// TwinCAT 3 PLC project Tc3_Handler
// ProgramVersion: 3.1.4024.0
// libraries:
//   Tc2_Standard, * (Beckhoff Automation GmbH)
//   Tc2_System, * (Beckhoff Automation GmbH)
//   Tc2_Utilities, * (Beckhoff Automation GmbH)
//   Tc3_Module, * (Beckhoff Automation GmbH)
// project tree:
//   / GVL.TcGVL (not stored), PlcTask.TcTTO
//   Library/Event/ E_Event.TcDUT, FB_Event.TcPOU, I_Event.TcIO, ST_Event.TcDUT
//   Library/Handler/ FB_Handler.TcPOU, I_Handler.TcIO
//   POUs/ FB_EventHandler.TcPOU, FB_EmergencyHandler.TcPOU, MAIN.TcPOU
// real-time tasks:
//   TASK PlcTask: cycle T#10ms, priority 20, ADS port 350

CONFIGURATION Tc3_Handler
    RESOURCE PLC ON TwinCAT3
        TASK PlcTask(INTERVAL := T#10ms, PRIORITY := 20);
        PROGRAM MAIN WITH PlcTask : MAIN;
    END_RESOURCE
END_CONFIGURATION

// ---- Library/Event/E_Event.TcDUT
{attribute 'qualified_only'}
{attribute 'strict'}
TYPE E_Event :
(
	Debug		:= 0,
	Info		:= 1,
    Warning		:= 2,
    Error		:= 3
)USINT;
END_TYPE

// ---- Library/Event/ST_Event.TcDUT
TYPE ST_Event :
STRUCT
	bEvent:		BOOL;
	bActive:	BOOL;
	eEvent:		E_Event;
	nTimestamp:	ULINT;
	nID:		DINT;
	sMessage:	STRING(255);
	sArguments:	STRING(255);
	sDefault:	STRING(255);
END_STRUCT
END_TYPE

// ---- Library/Event/I_Event.TcIO
INTERFACE I_Event

END_INTERFACE

// ---- Library/Handler/I_Handler.TcIO
INTERFACE I_Handler

METHOD PUBLIC M_Request
VAR_INPUT
	stEvent:			ST_Event;
END_VAR
END_METHOD

PROPERTY PUBLIC P_Next : I_Handler
GET
END_GET
SET
END_SET
END_PROPERTY

END_INTERFACE

// ---- POUs/MAIN.TcPOU
PROGRAM MAIN
VAR
	fbEvent:				FB_Event;
	fbEventHandler:			FB_EventHandler;
	fbTcLoggerHandler:		FB_TcLoggerHandler;	
	fbEmergencyHandler:		FB_EmergencyHandler;
	bInit:					BOOL:= TRUE;
	bDebug:					BOOL;
	bInfo:					BOOL;
	bWarning: 				BOOL;
	bError: 				BOOL;
END_VAR

IF bInit THEN
	bInit:= FALSE;
	fbEvent.P_Handler:= fbEventHandler;
	fbEventHandler.P_Next:= fbEmergencyHandler;
	fbEmergencyHandler.P_Next:= fbTcLoggerHandler;
END_IF

fbEvent();
fbEventHandler();
fbTcLoggerHandler();
fbEmergencyHandler();

IF bDebug THEN
	fbEvent.M_Debug('Debug',1);
END_IF

IF bInfo THEN
	fbEvent.M_Info('Warning',2);
END_IF

IF bWarning THEN
	fbEvent.M_Warning('Warning',3);
END_IF

IF bError THEN
	fbEvent.M_Error('Emergency Stop', 4);
END_IF

END_PROGRAM

// ---- Library/Event/FB_Event.TcPOU
FUNCTION_BLOCK FB_Event IMPLEMENTS I_Event
VAR_INPUT
END_VAR
VAR_OUTPUT
END_VAR
VAR
	iHandler:			I_Handler;
	stDebug:			ST_Event;
	stInfo:				ST_Event;
	stWarning:			ST_Event;
	stError:			ST_Event;
END_VAR

IF stDebug.bActive THEN
	stDebug.bActive:= FALSE;
ELSE
	stDebug.nTimestamp:= 0;
END_IF

IF stInfo.bActive THEN
	stInfo.bActive:= FALSE;	
ELSE
	stInfo.nTimestamp:= 0;		
END_IF

IF stWarning.bActive THEN
	stWarning.bActive:= FALSE;	
ELSE
	stWarning.nTimestamp:= 0;	
END_IF

IF stError.bActive THEN
	stError.bActive:= FALSE;	
ELSE
	stError.nTimestamp:= 0;	
END_IF

METHOD PUBLIC M_Debug
VAR_INPUT
	sMessage:	STRING(255);
	nID:		DINT;
END_VAR
stDebug.bActive:= TRUE;
stDebug.bEvent:= FALSE;
IF stDebug.sMessage <> sMessage THEN
	stDebug.bEvent:= TRUE;
END_IF
IF stDebug.nTimestamp = 0 THEN
	stDebug.nTimestamp:= F_GetSystemTime();
	stDebug.bEvent:= TRUE;
END_IF
stDebug.eEvent:= E_Event.Debug;
stDebug.sMessage:= sMessage;
stDebug.nID:= nID;

IF iHandler <> 0 THEN
	iHandler.M_Request(stDebug);
END_IF
END_METHOD

METHOD PUBLIC M_Error
VAR_INPUT
	sMessage:	STRING(255);
	nID:		DINT;
END_VAR
stError.bActive:= TRUE;
stError.bEvent:= FALSE;
IF stError.sMessage <> sMessage THEN
	stError.bEvent:= TRUE;
END_IF
IF stError.nTimestamp = 0 THEN
	stError.nTimestamp:= F_GetSystemTime();
	stError.bEvent:= TRUE;
END_IF
stError.eEvent:= E_Event.Error;
stError.sMessage:= sMessage;
stError.nID:= nID;

IF iHandler <> 0 THEN
	iHandler.M_Request(stError);
END_IF
END_METHOD

METHOD PUBLIC M_Info
VAR_INPUT
	sMessage:	STRING(255);
	nID:		DINT;
END_VAR
stInfo.bActive:= TRUE;
stInfo.bEvent:= FALSE;
IF stInfo.sMessage <> sMessage THEN
	stInfo.bEvent:= TRUE;
END_IF
IF stInfo.nTimestamp = 0 THEN
	stInfo.nTimestamp:= F_GetSystemTime();
	stInfo.bEvent:= TRUE;
END_IF
stInfo.eEvent:= E_Event.Info;
stInfo.sMessage:= sMessage;
stInfo.nID:= nID;

IF iHandler <> 0 THEN
	iHandler.M_Request(stInfo);
END_IF
END_METHOD

METHOD M_Warning
VAR_INPUT
	sMessage:	STRING(255);
	nID:		DINT;
END_VAR
stWarning.bActive:= TRUE;
stWarning.bEvent:= FALSE;
IF stWarning.sMessage <> sMessage THEN
	stWarning.bEvent:= TRUE;
END_IF
IF stWarning.nTimestamp = 0 THEN
	stWarning.nTimestamp:= F_GetSystemTime();
	stWarning.bEvent:= TRUE;
END_IF
stWarning.eEvent:= E_Event.Warning;
stWarning.sMessage:= sMessage;
stWarning.nID:= nID;

IF iHandler <> 0 THEN
	iHandler.M_Request(stWarning);
END_IF
END_METHOD

PROPERTY PUBLIC P_Handler : I_Handler
GET
P_Handler:= iHandler;
END_GET
SET
iHandler:= P_Handler;
END_SET
END_PROPERTY

END_FUNCTION_BLOCK

// ---- POUs/FB_EventHandler.TcPOU
FUNCTION_BLOCK FB_EventHandler EXTENDS FB_Handler
VAR_INPUT
END_VAR
VAR_OUTPUT
	bDebug:			BOOL;
	bInfo:			BOOL;
	bWarning:		BOOL;
	bError:			BOOL;
END_VAR
VAR
	nLength:		INT;
	aEvents:		ARRAY [0..100] OF ST_Event;
	nIndex: 		INT;
END_VAR

SUPER^();
nIndex:= 0;
WHILE nIndex < nLength DO
	IF aEvents[nIndex].bActive THEN
		aEvents[nIndex].bActive:= FALSE;
	ELSE
		M_Remove(nIndex);
	END_IF
	nIndex := nIndex + 1;
END_WHILE
bDebug:= FALSE;
bInfo:= FALSE;
bWarning:= FALSE;
bError:= FALSE;

METHOD PRIVATE M_Find : INT
VAR_INPUT
	stEvent:			ST_Event;		// event to find
END_VAR
M_Find := -1;
nIndex:= 0;
WHILE nIndex < nLength DO
    IF aEvents[nIndex].eEvent = stEvent.eEvent AND_THEN aEvents[nIndex].sMessage = stEvent.sMessage THEN
        M_Find := nIndex;
        RETURN;
    END_IF
	nIndex := nIndex + 1;
END_WHILE
END_METHOD

METHOD PRIVATE M_Remove
VAR_INPUT
	nPosition:			INT;
END_VAR
memcpy(ADR(aEvents[nIndex]), ADR(aEvents[nPosition + 1]), (SIZEOF(ST_Event) * (100  - nPosition)));
nLength:= nLength - 1;
END_METHOD

METHOD PUBLIC M_Request
VAR_INPUT
	stEvent:			ST_Event;		// event to be handled. 
END_VAR
VAR
	nFind:				INT;
END_VAR
// Update list
IF nLength < 100 THEN
	nFind:= M_Find(stEvent);
	IF nFind = -1 THEN
		aEvents[nLength]:= stEvent;
		nLength:= nLength + 1;
	ELSE
		aEvents[nFind]:= stEvent;		
	END_IF
END_IF

// Update outputs
CASE stEvent.eEvent OF
	E_Event.Debug:
		bDebug:= TRUE;
	E_Event.Info:
		bInfo:= TRUE;
	E_Event.Warning:
		bWarning:= TRUE;
	E_Event.Error:
		bError:= TRUE;
END_CASE

// Update Logger
IF stEvent.bEvent THEN
	CASE stEvent.eEvent OF
		E_Event.Debug:
			ADSLOGSTR(ADSLOG_MSGTYPE_HINT OR ADSLOG_MSGTYPE_LOG, stEvent.sMessage, '');
		E_Event.Info:
			ADSLOGSTR(ADSLOG_MSGTYPE_HINT OR ADSLOG_MSGTYPE_LOG, stEvent.sMessage, '');
		E_Event.Warning:
			ADSLOGSTR(ADSLOG_MSGTYPE_WARN OR ADSLOG_MSGTYPE_LOG, stEvent.sMessage, '');
		E_Event.Error:
			ADSLOGSTR(ADSLOG_MSGTYPE_ERROR OR ADSLOG_MSGTYPE_LOG, stEvent.sMessage, '');
	END_CASE
END_IF

SUPER^.M_Request(stEvent);
END_METHOD

END_FUNCTION_BLOCK

// ---- Library/Handler/FB_Handler.TcPOU
FUNCTION_BLOCK ABSTRACT FB_Handler IMPLEMENTS I_Handler
VAR_INPUT
END_VAR
VAR_OUTPUT
END_VAR
VAR
	iHandler:			I_Handler;
END_VAR

//	The FB_Handler is an abstract function block that implements the I_Handler interface. 
//	It represents a handler in the Chain of Responsibility pattern,
//	where a request can be passed along a chain of potential handlers until one of them handles the request.
//	Each handler in the chain has the ability to either handle the request or pass it to the next handle

METHOD PUBLIC M_Request
VAR_INPUT
	stEvent:			ST_Event;		// event to be handled. 
END_VAR
// The M_Request method is used to handle the request.

IF iHandler <> 0 THEN
	// the request is passed to the next handler 
	iHandler.M_Request(stEvent);
END_IF
END_METHOD

PROPERTY PUBLIC P_Next : I_Handler
GET
P_Next:= iHandler;
END_GET
SET
iHandler:= P_Next;
END_SET
END_PROPERTY

END_FUNCTION_BLOCK

// ---- POUs/FB_EmergencyHandler.TcPOU
FUNCTION_BLOCK FB_EmergencyHandler EXTENDS FB_Handler
VAR_INPUT
	bReset:			BOOL;
END_VAR
VAR_OUTPUT
	bOutput:		BOOL;
END_VAR
VAR
	bResetOld: 		BOOL:= TRUE;
END_VAR

SUPER^();
IF bReset AND NOT bResetOld THEN
	bOutput:= TRUE;
END_IF
bResetOld:= bReset;

METHOD PUBLIC M_Request
VAR_INPUT
	stEvent:			ST_Event;		// event to be handled. 
END_VAR
IF stEvent.sMessage = 'Emergency Stop' THEN
	bOutput:= FALSE;
END_IF

SUPER^.M_Request(stEvent);
END_METHOD

END_FUNCTION_BLOCK
